TYPE OutputSignals :
STRUCT
	Motor1 : INT; // 1 is forward motion, -1 is backward motion, 0 standstill
	Motor2 : INT;  // 1 is counterclockwise rotation, -1 is clockwise rotation, 0 standstill
	GripperMotor : INT; // 1 is lift, -1 is lower, 0 is standstill
	Gripper : BOOL := TRUE; // TRUE when gripper open, FALSE when gripper is closed
	// The above selection of values is indicative, and not actually signals that will be send to the Motors. The values just show 
	// whether a motor is energized (zero or non-zero) and in which direction is energized (-1, 1) in order to showcase forward or reverse direction of motor rotation
END_STRUCT
END_TYPE

(* stored: Version 1.1.0.1, ProductVersion 3.1.4024.12
   DUT OutputSignals: Id {dafb8af1-1675-48b1-ba91-f7b6edc27966} *)
